IF NOT (Transfer.Mode = FIT_VFD_Transfer_Modes.Pause) AND NOT (Transfer.Mode = FIT_VFD_Transfer_Modes.Resume) THEN _w1 := Transfer.Mode; END_IF
Transfer.cONFIG.Mode_Memory := _w1;
IF Transfer.Mode = FIT_VFD_Transfer_Modes.Resume THEN _w2 := Transfer.Config.Mode_Memory; END_IF
Transfer.Mode := _w2;
Transfer.Status := SEL(VFD_Not_Ready, SEL(BCV_Not_Ready, SEL(ACV_Not_Ready, SEL(Transfer.Mode=FIT_VFD_Transfer_Modes.Lock_Out, SEL(False, SEL(Complete, SEL(Transfer_Running, SEL(FIT.PLC_Reset, SEL(IDLE_Return, SEL(PAUSED, Transfer_status.IDLE, Transfer_status.Paused), Transfer_status.IDLE), Transfer_status.FIT_Reset), Transfer_status.Running), Transfer_status.Complete), Transfer_status.Complete), Transfer_status.LOCKED_OUT), Transfer_status.ACV_Not_Ready), Transfer_status.BCV_Not_Ready), Transfer_status.VFD_Not_Ready);
_w3 := Transfer.Mode = FIT_VFD_Transfer_Modes.Idle;
_w4 := True AND NOT (BCV.Status = Burkert.eBCV_Status.A_Closed);
BCV_Not_Ready := _w3 AND _w4;
_w5 := True AND NOT (VFD.MODE.eMode = eVFD_Modes.Auto);
_w6 := _w4 OR _w5;
SR2(SET1 := _w3 AND _w6, RESET := NOT _w6); // SR
IF SR2.Q1 THEN _w7 := FIT_VFD_Transfer_Modes.Idle; END_IF
Transfer.Mode := _w7;
VFD_Not_Ready := _w3 AND _w5;
_w8 := Transfer.Status = Transfer_Status.Complete;
_w9 := Transfer.Status = Transfer_Status.BCV_Not_Ready OR Transfer.Status = Transfer_Status.VFD_Not_Ready;
_w10 := Transfer_Status.IDLE = Transfer.Status OR False OR Transfer.Status = Transfer_Status.LOCKED_OUT;
_w11 := Transfer.Mode = FIT_VFD_Transfer_Modes.Pause;
PAUSED := _w11;
_w12 := Transfer.Mode = FIT_VFD_Transfer_Modes.IDLE;
_w13 := Complete OR Error OR _w12 OR _w11;
_w14 := NOT Pump_Start OR _w13;
CTRL_PID_1(
    ACT := FIT.Rate,
    SET := Transfer.Config.Target_Rate,
    SUP := 0.0,
    OFS := Transfer.Config.Target_Rate * Transfer.Config.FF,
    M_I := 0.0,
    MAN := _w14,
    RST := _w14,
    KP := Transfer.Config.KP,
    TN := Transfer.Config.TN,
    TV := Transfer.Config.TV,
    LL := 0,
    LH := 100); // BURKERT_OSCAT_BASIC.CTRL_PID
PID_CV := CTRL_PID_1.Y;
TP11(IN := NOT LockOut_Active AND _w13, PT := t#5s); // TP
VFD.PLC_Run := SEL(TP11.Q, VFD.PLC_Run, FALSE);
VFD.PLC_CMD := SEL(TP11.Q, VFD.PLC_CMD, 0.0);
F_TRIG_0(CLK := TP11.Q); // F_Trig
BCV.PLC_CMD := SEL(F_TRIG_0.Q, BCV.PLC_CMD, False);
IDLE_Return := _w9 AND _w12;
SR_10(SET1 := FIT.Total<1, RESET := _w12); // SR
TON_10(IN := SR_10.Q1, PT := T#2s); // TON
FIT_Reset_Complete := TON_10.Q;
R_TRIG_0(CLK := _w12 OR TON_10.Q); // R_trig
_w15 := SEL(R_TRIG_0.Q, FIT.PLC_Reset, False);
_w16 := Transfer.Mode = FIT_VFD_Transfer_Modes.Batch;
_w17 := False OR False OR _w16;
Flow_Mode := _w17;
_w18 := _w17 AND FIT_Reset_Complete AND NOT Complete AND NOT Error AND NOT Time_Complete;
Transfer_Running := _w18;
transfer.Remaining_Volume := SEL(_w18, 0, Transfer.Config.Target_Volume-fit.Total);
_w19 := True AND _w18;
Enable_Pump := _w19;
BCV.PLC_CMD := SEL(_w19, BCV.PLC_CMD, TRUE);
_w20 := _w16 AND FIT_Reset_Complete AND FIT.Total >= Transfer.Config.Target_Volume;
Batch_Complete := _w20;
RS_11(SET := Time_Complete OR _w20 OR False, RESET1 := _w12); // RS
Complete := RS_11.Q1;
_w21 := LOCK_OUT AND _w10 AND NOT RS_11.Q1;
F_TRIG_10(CLK := _w21); // F_Trig
IF F_TRIG_10.Q THEN _w22 := FIT_VFD_Transfer_Modes.Idle; END_IF
Transfer.Mode := _w22;
_w23 := _w21;
IF _w23 THEN _w24 := FIT_VFD_Transfer_Modes.Lock_Out; END_IF
LockOut_Active := _w23;
Transfer.Mode := _w24;
FIT.PLC_Reset := SEL(NOT SR_10.Q1 AND _w17 AND NOT _w20, _w15, True);
_w25 := SEL(_w19, _w18, BCV.Status = Burkert.eBCV_Status.A_Open);
Pump_Start := _w25;
_w26 := SEL(_w25, VFD.PLC_CMD, PID_CV);
Transfer.Config.Motor_PCT := _w26;
VFD.PLC_CMD := _w26;
VFD.PLC_Run := SEL(_w25, VFD.PLC_Run, PID_CV > 15);
TON_12(IN := _w8, PT := T#10s); // TON

END_FUNCTION_BLOCK

// 25 Interfaces/IcSensorProvider
INTERFACE IcSensorProvider:

END_INTERFACE;

METHOD GetSensorRef : POINTER TO Burkert.cSensor
VAR_INPUT
        eSensor : cSensor_Mapping;
END_VAR
END_METHOD

END_INTERFACE

// 50 Functions/DaySeconds
FUNCTION DaySeconds : UDINT
VAR_INPUT
	Hour:UINT;
	Minute:UINT;
	Second:UINT;
END_VAR
VAR
END_VAR

(* body of a kind this reader does not render *)

END_FUNCTION

// GetLibVersion
// This function has been automatically generated from the project information.
FUNCTION GetLibVersion : VERSION
VAR_INPUT
	
END_VAR

GetLibVersion.uiMajor := 3;
GetLibVersion.uiMinor := 0;
GetLibVersion.uiServicePack := 0;
GetLibVersion.uiPatch := 49;

END_FUNCTION

// GetLibVersionNumber
// This function has been automatically generated from the project information.
FUNCTION GetLibVersionNumber : DWORD
VAR_INPUT
	
END_VAR

GetLibVersionNumber := 50331697;

END_FUNCTION

// IsLibReleased
// This function has been automatically generated from the project information.
FUNCTION IsLibReleased : BOOL
VAR_INPUT
	
END_VAR

IsLibReleased := FALSE;

END_FUNCTION

// GetBooleanProperty
// This function has been automatically generated from the project information.
{attribute 'signature_flag' := '1073741824'}
{attribute 'register_in_runtime'}
FUNCTION GetBooleanProperty : BOOL
VAR_INPUT
	stKey: WSTRING;
END_VAR

IF stKey = "IsEndUserLibrary" THEN
	GetBooleanProperty := FALSE;
ELSIF stKey = "IsStorageFormatPinned" THEN
	GetBooleanProperty := FALSE;
ELSIF stKey = "Released" THEN
	GetBooleanProperty := FALSE;
ELSE
	GetBooleanProperty := FALSE;
END_IF

END_FUNCTION

// GetCompany
// This function has been automatically generated from the project information.
{attribute 'signature_flag' := '1073741824'}
{attribute 'register_in_runtime'}
FUNCTION GetCompany : WSTRING
VAR_INPUT
	
END_VAR

GetCompany := "Burkert-Canada";

END_FUNCTION

// GetTextProperty2
// This function has been automatically generated from the project information.
{attribute 'signature_flag' := '1073741824'}
{attribute 'register_in_runtime'}
FUNCTION GetTextProperty2 : POINTER TO WSTRING
VAR_INPUT
	stKey: WSTRING;
END_VAR

IF stKey = "Author" THEN
	GetTextProperty2 := ADR("Robert Budgen");
ELSIF stKey = "Company" THEN
	GetTextProperty2 := ADR("Burkert-Canada");
ELSIF stKey = "CompiledLibraryCompatibilityVersion" THEN
	GetTextProperty2 := ADR("e!COCKPIT");
ELSIF stKey = "DefaultNamespace" THEN
	GetTextProperty2 := ADR("Brau");
ELSIF stKey = "Description" THEN
	GetTextProperty2 := ADR("");
ELSIF stKey = "LanguageModelAttribute" THEN
	GetTextProperty2 := ADR("qualified-access-only");
ELSIF stKey = "Placeholder" THEN
	GetTextProperty2 := ADR("Brau");
ELSIF stKey = "Project" THEN
	GetTextProperty2 := ADR("Burkert Canada");
ELSIF stKey = "Title" THEN
	GetTextProperty2 := ADR("Brau");
ELSE
	GetTextProperty2 := ADR("");
END_IF

END_FUNCTION

// GetTextProperty
// This function has been automatically generated from the project information.
{attribute 'signature_flag' := '1073741824'}
{attribute 'register_in_runtime'}
FUNCTION GetTextProperty : WSTRING
VAR_INPUT
	stKey: WSTRING;
END_VAR

IF stKey = "Author" THEN
	GetTextProperty := "Robert Budgen";
ELSIF stKey = "Company" THEN
	GetTextProperty := "Burkert-Canada";
ELSIF stKey = "CompiledLibraryCompatibilityVersion" THEN
	GetTextProperty := "e!COCKPIT";
ELSIF stKey = "DefaultNamespace" THEN
	GetTextProperty := "Brau";
ELSIF stKey = "Description" THEN
	GetTextProperty := "";
ELSIF stKey = "LanguageModelAttribute" THEN
	GetTextProperty := "qualified-access-only";
ELSIF stKey = "Placeholder" THEN
	GetTextProperty := "Brau";
ELSIF stKey = "Project" THEN
	GetTextProperty := "Burkert Canada";
ELSIF stKey = "Title" THEN
	GetTextProperty := "Brau";
ELSE
	GetTextProperty := "";
END_IF

END_FUNCTION

// GetTitle
// This function has been automatically generated from the project information.
{attribute 'signature_flag' := '1073741824'}
{attribute 'register_in_runtime'}
FUNCTION GetTitle : WSTRING
VAR_INPUT
	
END_VAR

GetTitle := "Brau";

END_FUNCTION

// GetVersion
// This function has been automatically generated from the project information.
{attribute 'signature_flag' := '1073741824'}
{attribute 'register_in_runtime'}
FUNCTION GetVersion : VERSION
VAR_INPUT
	
END_VAR

GetVersion.uiMajor := 3;
GetVersion.uiMinor := 0;
GetVersion.uiServicePack := 0;
GetVersion.uiPatch := 49;

END_FUNCTION

// GetVersionProperty
// This function has been automatically generated from the project information.
{attribute 'signature_flag' := '1073741824'}
{attribute 'register_in_runtime'}
FUNCTION GetVersionProperty : VERSION
VAR_INPUT
	stKey: WSTRING;
END_VAR

IF stKey = "Version" THEN
	GetVersionProperty.uiMajor := 3;
	GetVersionProperty.uiMinor := 0;
	GetVersionProperty.uiServicePack := 0;
	GetVersionProperty.uiPatch := 49;
ELSE
	GetVersionProperty.uiMajor := 0;
	GetVersionProperty.uiMinor := 0;
	GetVersionProperty.uiServicePack := 0;
	GetVersionProperty.uiPatch := 0;
END_IF

END_FUNCTION

// Asi/AC2916_AIT
FUNCTION_BLOCK AC2916_AIT
VAR_INPUT
	//Raw:	REAL;
	LAS:BOOL:=TRUE;
	LDS:BOOL:=TRUE;
	LPS:BOOL:=TRUE;
	LPF:BOOL:=FALSE;
	Alarm_Enable:BOOL:=TRUE;
	Latching:BOOL:=FALSE;
	//Fault:BOOL:=FALSE;
	Online:BOOL:=TRUE;
	Raw:WORD;
END_VAR

VAR_OUTPUT
	//Status	:BYTE;
END_VAR
VAR_IN_OUT
AIT	:	Burkert.cAIT;
END_VAR

VAR
	hihi: BOOL;
	hi: BOOL;
	lolo: BOOL;
	LO: BOOL;
	Alarm_Debounce: TON;
	deboune_Time: TIME;
	Alarm_Active: BOOL;
	Alarm_Debounce_ET: TIME;
	Alarm: BOOL;
	ALARM_2_0: BURKERT_OSCAT_BASIC.ALARM_2;
	F_TRIG_0: F_Trig;
	TON_0: TON;
	tmpEU: REAL;
	//tmpEU1: REAL;
	tmpEU2: REAL;
END_VAR

VAR_TEMP
	EU_Range: REAL;
	Raw_Range: REAL;
	Corrected_Raw: REAL;
	Raw_Pct: REAL;
	EU_Scaled: REAL;
END_VAR
VAR // added by the converter: edge detectors and wires of the graphical bodies
    _w1, _w2, _w3 : BOOL;
END_VAR

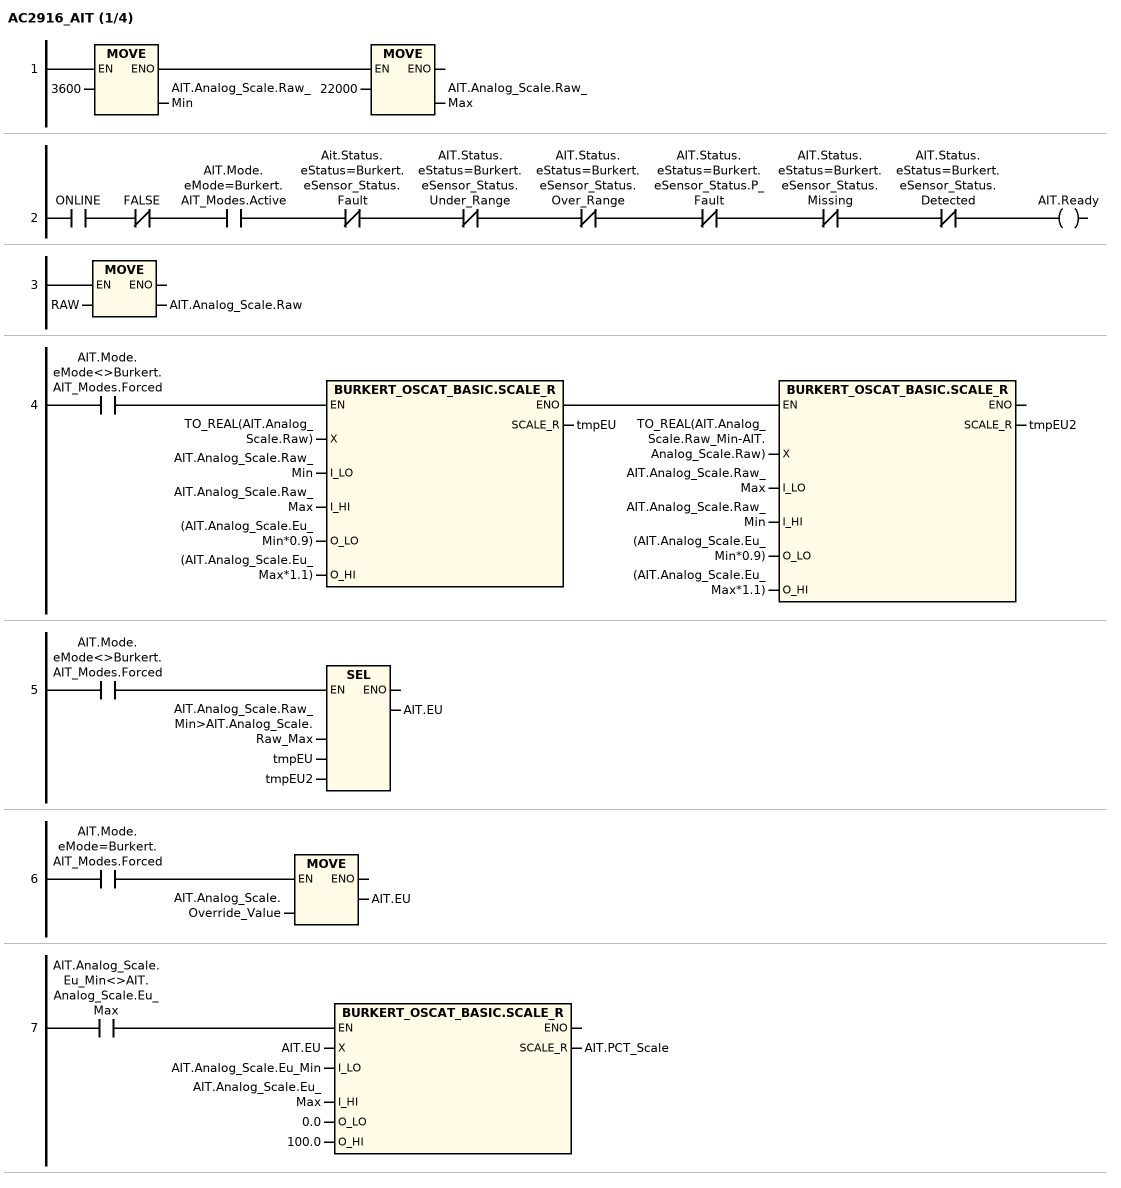
// NETWORK 1
AIT.Analog_Scale.Raw_Min := 3600;
AIT.Analog_Scale.Raw_Max := 22000;

// NETWORK 2
AIT.Ready := ONLINE AND NOT FALSE AND (AIT.Mode.eMode=Burkert.AIT_Modes.Active) AND NOT (Ait.Status.eStatus=Burkert.eSensor_Status.Fault) AND NOT (AIT.Status.eStatus=Burkert.eSensor_Status.Under_Range) AND NOT (AIT.Status.eStatus=Burkert.eSensor_Status.Over_Range) AND NOT (AIT.Status.eStatus=Burkert.eSensor_Status.P_Fault) AND NOT (AIT.Status.eStatus=Burkert.eSensor_Status.Missing) AND NOT (AIT.Status.eStatus=Burkert.eSensor_Status.Detected);

// NETWORK 3
AIT.Analog_Scale.Raw := RAW;

// NETWORK 4
_w1 := AIT.Mode.eMode<>Burkert.AIT_Modes.Forced;
IF _w1 THEN
    tmpEU := BURKERT_OSCAT_BASIC.SCALE_R(X := TO_REAL(AIT.Analog_Scale.Raw), I_LO := AIT.Analog_Scale.Raw_Min, I_HI := AIT.Analog_Scale.Raw_Max, O_LO := (AIT.Analog_Scale.Eu_Min*0.9), O_HI := (AIT.Analog_Scale.Eu_Max*1.1));
END_IF
IF _w1 THEN
    tmpEU2 := BURKERT_OSCAT_BASIC.SCALE_R(X := TO_REAL(AIT.Analog_Scale.Raw_Min-AIT.Analog_Scale.Raw), I_LO := AIT.Analog_Scale.Raw_Max, I_HI := AIT.Analog_Scale.Raw_Min, O_LO := (AIT.Analog_Scale.Eu_Min*0.9), O_HI := (AIT.Analog_Scale.Eu_Max*1.1));
END_IF

// NETWORK 5
IF AIT.Mode.eMode<>Burkert.AIT_Modes.Forced THEN
    AIT.EU := SEL(AIT.Analog_Scale.Raw_Min>AIT.Analog_Scale.Raw_Max, tmpEU, tmpEU2);
END_IF

// NETWORK 6
IF AIT.Mode.eMode=Burkert.AIT_Modes.Forced THEN AIT.EU := AIT.Analog_Scale.Override_Value; END_IF

// NETWORK 7
IF AIT.Analog_Scale.Eu_Min<>AIT.Analog_Scale.Eu_Max THEN
    AIT.PCT_Scale := BURKERT_OSCAT_BASIC.SCALE_R(X := AIT.EU, I_LO := AIT.Analog_Scale.Eu_Min, I_HI := AIT.Analog_Scale.Eu_Max, O_LO := 0.0, O_HI := 100.0);
END_IF

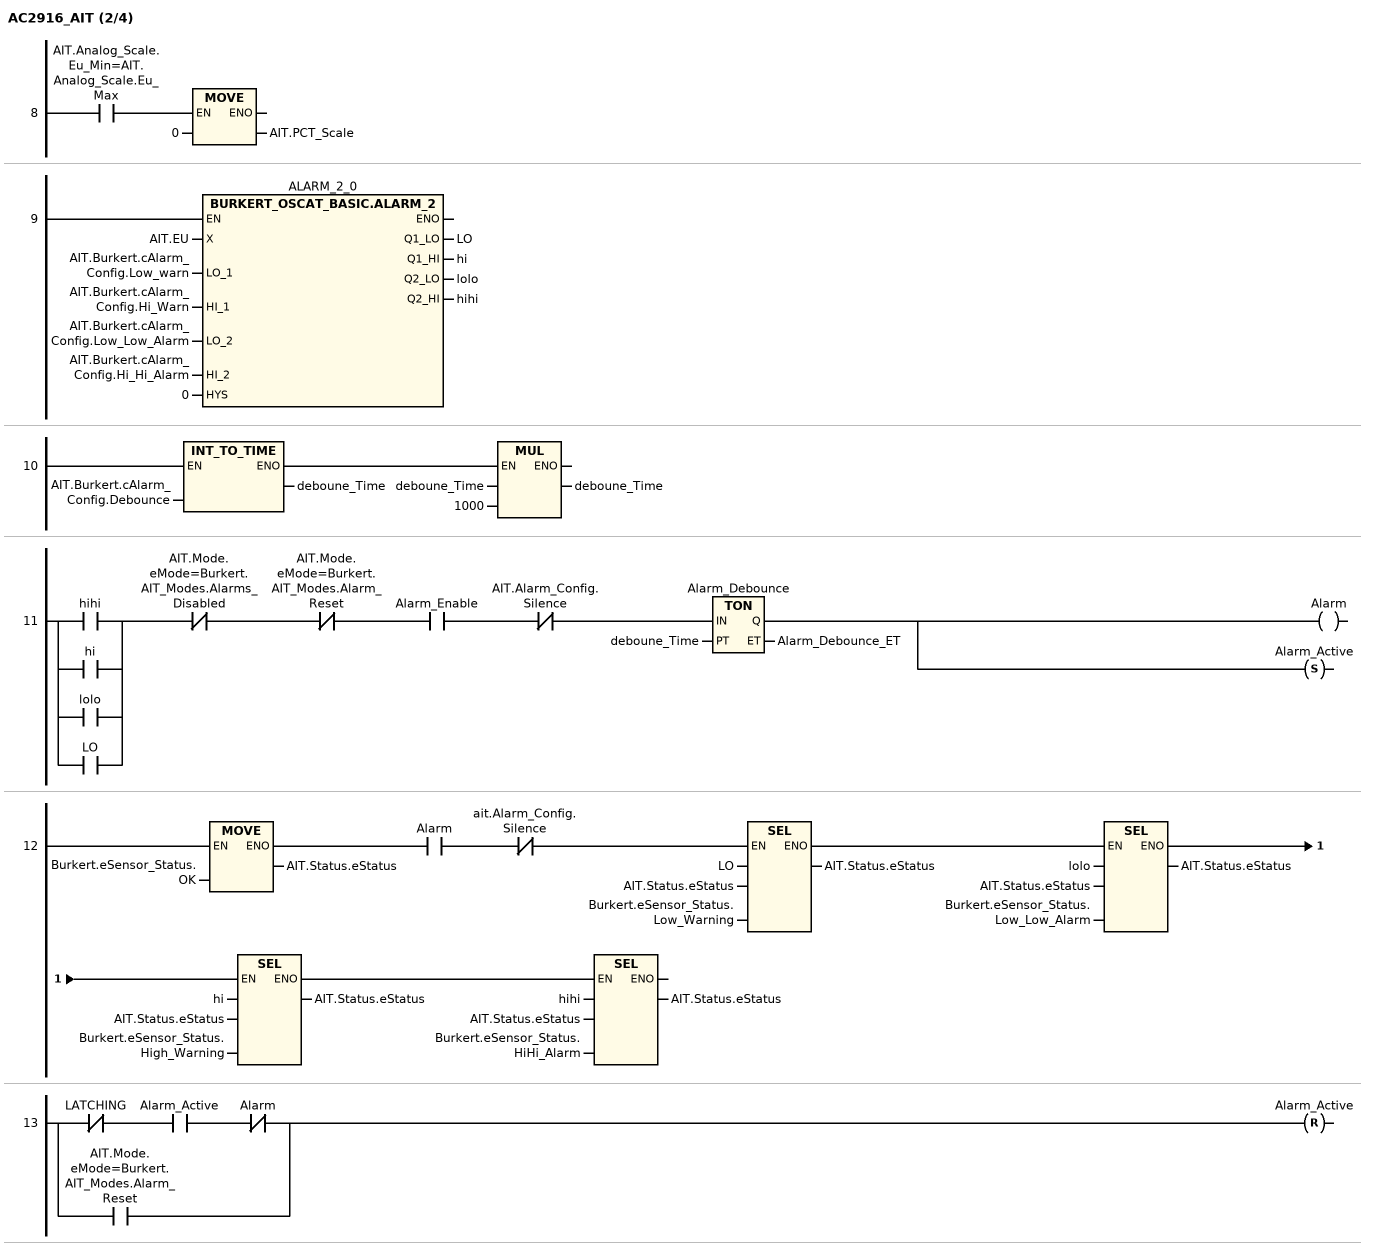
// NETWORK 8
IF AIT.Analog_Scale.Eu_Min=AIT.Analog_Scale.Eu_Max THEN AIT.PCT_Scale := 0; END_IF

// NETWORK 9
ALARM_2_0(
    X := AIT.EU,
    LO_1 := AIT.Burkert.cAlarm_Config.Low_warn,
    HI_1 := AIT.Burkert.cAlarm_Config.Hi_Warn,
    LO_2 := AIT.Burkert.cAlarm_Config.Low_Low_Alarm,
    HI_2 := AIT.Burkert.cAlarm_Config.Hi_Hi_Alarm,
    HYS := 0,
    Q1_LO => LO,
    Q1_HI => hi,
    Q2_LO => lolo,
    Q2_HI => hihi); // BURKERT_OSCAT_BASIC.ALARM_2

// NETWORK 10
deboune_Time := INT_TO_TIME(AIT.Burkert.cAlarm_Config.Debounce);
deboune_Time := deboune_Time * 1000;

// NETWORK 11
Alarm_Debounce(
    IN := (hihi OR hi OR lolo OR LO) AND NOT (AIT.Mode.eMode=Burkert.AIT_Modes.Alarms_Disabled) AND NOT (AIT.Mode.eMode=Burkert.AIT_Modes.Alarm_Reset) AND Alarm_Enable AND NOT AIT.Alarm_Config.Silence,
    PT := deboune_Time,
    ET => Alarm_Debounce_ET); // TON
Alarm := Alarm_Debounce.Q;
Alarm_Active S= Alarm_Debounce.Q;

// NETWORK 12
AIT.Status.eStatus := Burkert.eSensor_Status.OK;
_w2 := Alarm AND NOT ait.Alarm_Config.Silence;
IF _w2 THEN AIT.Status.eStatus := SEL(LO, AIT.Status.eStatus, Burkert.eSensor_Status.Low_Warning); END_IF
IF _w2 THEN AIT.Status.eStatus := SEL(lolo, AIT.Status.eStatus, Burkert.eSensor_Status.Low_Low_Alarm); END_IF
IF _w2 THEN AIT.Status.eStatus := SEL(hi, AIT.Status.eStatus, Burkert.eSensor_Status.High_Warning); END_IF
IF _w2 THEN AIT.Status.eStatus := SEL(hihi, AIT.Status.eStatus, Burkert.eSensor_Status.HiHi_Alarm); END_IF

// NETWORK 13
Alarm_Active R= NOT LATCHING AND Alarm_Active AND NOT Alarm OR (AIT.Mode.eMode=Burkert.AIT_Modes.Alarm_Reset);

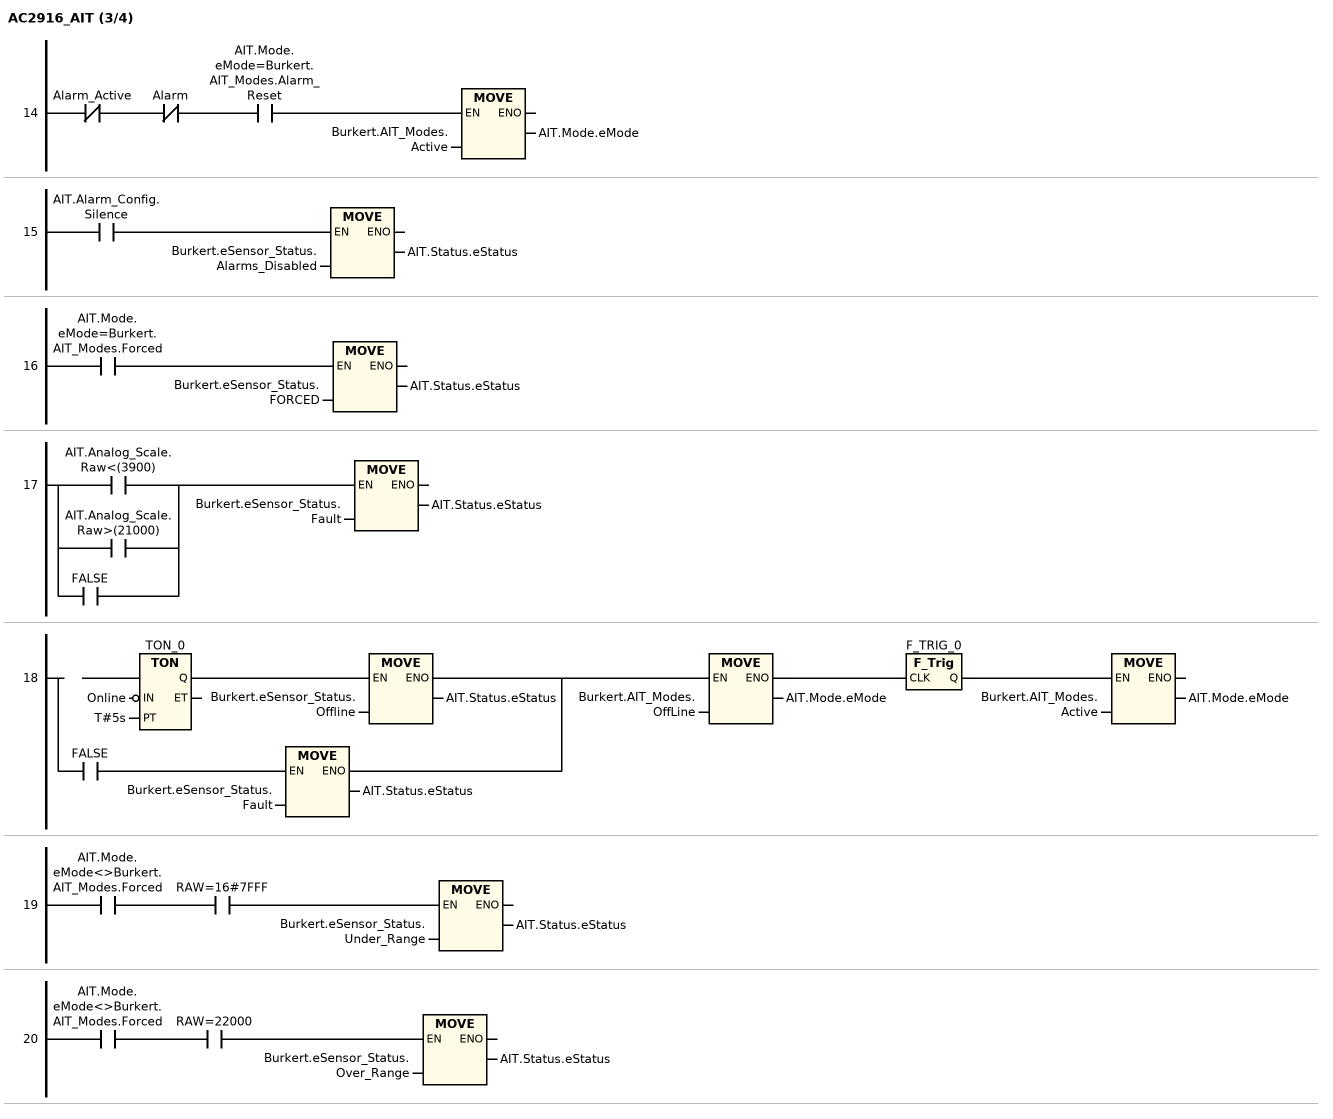
// NETWORK 14
IF NOT Alarm_Active AND NOT Alarm AND (AIT.Mode.eMode=Burkert.AIT_Modes.Alarm_Reset) THEN
    AIT.Mode.eMode := Burkert.AIT_Modes.Active;
END_IF

// NETWORK 15
IF AIT.Alarm_Config.Silence THEN AIT.Status.eStatus := Burkert.eSensor_Status.Alarms_Disabled; END_IF

// NETWORK 16
IF AIT.Mode.eMode=Burkert.AIT_Modes.Forced THEN AIT.Status.eStatus := Burkert.eSensor_Status.FORCED; END_IF

// NETWORK 17
IF (AIT.Analog_Scale.Raw<(3900)) OR (AIT.Analog_Scale.Raw>(21000)) OR FALSE THEN
    AIT.Status.eStatus := Burkert.eSensor_Status.Fault;
END_IF

// NETWORK 18
TON_0(IN := NOT Online, PT := T#5s); // TON
_w3 := TON_0.Q;
IF _w3 THEN AIT.Status.eStatus := Burkert.eSensor_Status.Offline; END_IF
IF FALSE THEN AIT.Status.eStatus := Burkert.eSensor_Status.Fault; END_IF
IF _w3 OR FALSE THEN AIT.Mode.eMode := Burkert.AIT_Modes.OffLine; END_IF
F_TRIG_0(CLK := _w3 OR FALSE); // F_Trig
IF F_TRIG_0.Q THEN AIT.Mode.eMode := Burkert.AIT_Modes.Active; END_IF

// NETWORK 19
IF (AIT.Mode.eMode<>Burkert.AIT_Modes.Forced) AND (RAW=16#7FFF) THEN
    AIT.Status.eStatus := Burkert.eSensor_Status.Under_Range;
END_IF

// NETWORK 20
IF (AIT.Mode.eMode<>Burkert.AIT_Modes.Forced) AND (RAW=22000) THEN
    AIT.Status.eStatus := Burkert.eSensor_Status.Over_Range;
END_IF

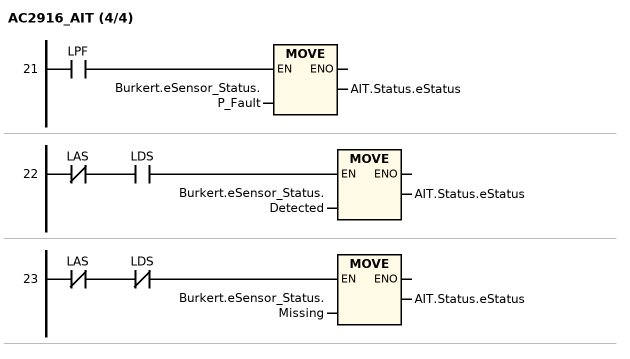
// NETWORK 21
IF LPF THEN AIT.Status.eStatus := Burkert.eSensor_Status.P_Fault; END_IF

// NETWORK 22
IF NOT LAS AND LDS THEN AIT.Status.eStatus := Burkert.eSensor_Status.Detected; END_IF

// NETWORK 23
IF NOT LAS AND NOT LDS THEN AIT.Status.eStatus := Burkert.eSensor_Status.Missing; END_IF

END_FUNCTION_BLOCK

// Asi/ACV_ASI_CTRL_UDFB
FUNCTION_BLOCK ACV_ASI_CTRL_UDFB
VAR_INPUT
	FB:INT;
	CutOff:REAL:=0;
	LOCKOUT:BOOL:=FALSE;
	Online:BOOL:=TRUE;
	Error_PCT:REAL:=10;
	Error_Delay_S:INT:=10;
	LAS:BOOL:=TRUE;
	LDS:BOOL:=TRUE;
	LPS:BOOL:=TRUE;
	LPF:BOOL:=FALSE;
END_VAR
VAR_OUTPUT
	Status	:INT;
	Output	:INT;
END_VAR
VAR_IN_OUT
	//Valve	:ACV_DUT;
END_VAR
VAR
	//Output_TMP: REAL;
	//Scaled_Out: REAL;
	TON_1: TON;
	TOF_0: TOF;
	tmp_Output: REAL;
	FB_Real: REAL;
	Burkert_mode: Ton;
END_VAR

VAR_IN_OUT
	Valve:Burkert.ASi_8694;
END_VAR

(* body of a kind this reader does not render *)

END_FUNCTION_BLOCK

// Asi/B8681_ASI_UDFB
FUNCTION_BLOCK B8681_ASI_UDFB
VAR_INPUT
	RX:BYTE;
	LAS:BOOL:=TRUE;
	LDS:BOOL:=TRUE;
	LPS:BOOL:=TRUE;
	LPF:BOOL:=FALSE;
END_VAR
VAR_OUTPUT
	TX:BYTE;
END_VAR
VAR
	lcl_status: BYTE;
END_VAR
VAR_IN_OUT
	Valve:Burkert.B8691_Asi_DUT;
END_VAR
VAR // added by the converter: edge detectors and wires of the graphical bodies
    _w1, _w2, _w3 : ANY;
END_VAR

_w1 := (Valve.Mode=Burkert.e_8681_Modes.Auto) AND (Valve.PLC_CMD=Burkert.e_8681_Modes.Upper_Drain) OR (Valve.Mode=Burkert.e_8681_Modes.Upper_Drain);
_w2 := SEL(_w1, SEL((Valve.Mode=Burkert.e_8681_Modes.Auto) AND (Valve.PLC_CMD=Burkert.e_8681_Modes.Lower_Drain) OR (Valve.Mode=Burkert.e_8681_Modes.Lower_Drain), SEL((Valve.Mode=Burkert.e_8681_Modes.Auto) AND (Valve.PLC_CMD=Burkert.e_8681_Modes.Open) OR (Valve.Mode=Burkert.e_8681_Modes.Open), 0, 1), 2), 4);
TX := _w2;
BURKERT_OSCAT_BASIC.WORD_OF_BYTE\(B1 := _w2, B0 := RX, WORD_OF_BYTE => _w3);
Valve.Status := _w3;
Valve.Status1 := SEL(LPF, SEL(LDS AND NOT LAS, SEL(NOT LAS, SEL(RX.2, SEL(_w1, SEL(RX.0, SEL(RX.1, eB8681_Status.Unknown, eB8681_Status.Open), eB8681_Status.Blocked), eB8681_Status.Upper_Drain), eB8681_Status.Lower_Drain), eB8681_Status.Missing), eB8681_Status.Detected), eB8681_Status.P_Fault);

END_FUNCTION_BLOCK

// Asi/BCV_ASI_CTRL_UDFB
FUNCTION_BLOCK BCV_ASI_CTRL_UDFB
VAR_INPUT
	OL:BOOL;
	CL:BOOL;
	LOCKOUT:BOOL:=FALSE;
	Online:BOOL:=TRUE;
	LAS:BOOL:=TRUE;
	LDS:BOOL:=TRUE;
	LPS:BOOL:=TRUE;
	LPF:BOOL:=FALSE;

END_VAR
VAR_OUTPUT
	Output	:BOOL;
END_VAR
VAR_IN_OUT
	BCV:Burkert.cBCV;
END_VAR
VAR
	
	Test: BOOL;
	GEN_PULSE_0: Burkert_OSCAT_BASIC.GEN_PULSE;
	Burkert_Open_Ton: TON;
END_VAR

(* body of a kind this reader does not render *)

END_FUNCTION_BLOCK

// Burkert Library/Parse_DDO
FUNCTION_BLOCK Parse_DDO
VAR_INPUT
	ORF_data:POINTER TO BYTE;
	Node:BYTE;
	Request_Size:INT:=10;
	
END_VAR
VAR_OUTPUT
	DDO:eDip_DDO;
END_VAR
VAR
	Block_Size:UINT;
	lcl_pointer:POINTER TO BYTE;
	DDO_Index:INT;
	ORF_Node:BYTE;
	ORF_Index_HB:BYTE;
	ORF_Index_LB:BYTE;
	ORF_SubIndex:BYTE;
	
	
END_VAR

Block_Size:=SIZEOF(ORF_Request);
lcl_pointer:=ORF_Data;

FOR DDO_Index := 0 TO Request_Size BY 1 DO
	
	ORF_Index_LB:=lcl_pointer[0];
	ORF_Index_HB:=LCL_Pointer[1];
	ORF_SubIndex:=lcl_pointer[2];
	ORF_Node:=lcl_pointer[3];
	
	
	IF (lcl_pointer[10]=1) AND (ORF_Node= Node) AND (ORF_Index_HB=16#20) AND (ORF_Index_LB=16#00) THEN
		MEMUtils.MemSet(pbyBuffer:=lcl_pointer+10 , byValue:=0 , dwSize:= 1); // Clear Complete
		CASE ORF_SubIndex OF
			16#02: //16#2000-2
				MEMUtils.MemCpy(pbyDest:=ADR(DDO.Ident)+2 , pbySrc:=lcl_pointer+4 , dwSize:=2 );
				MEMUtils.MemCpy(pbyDest:=ADR(DDO.Ident) , pbySrc:=lcl_pointer+6 , dwSize:=2 );
				lcl_pointer[9]:=BOOL_TO_BYTE(DDO.Ident=0);
				//MEMUtils.MemSet(pbyBuffer:=lcl_pointer+9 , byValue:=1 , dwSize:= 1);// Set Enable				
			16#07: //16#2000-7
				MEMUtils.MemCpy(pbyDest:=ADR(DDO.Serial)+2 , pbySrc:=lcl_pointer+4 , dwSize:=2 );
				MEMUtils.MemCpy(pbyDest:=ADR(DDO.Serial) , pbySrc:=lcl_pointer+6 , dwSize:=2 );
				lcl_pointer[9]:=BOOL_TO_BYTE(DDO.Serial=0);
			16#008: //16#2000-8
				MEMUtils.MemCpy(pbyDest:=ADR(DDO.Product_Code)+2 , pbySrc:=lcl_pointer+4 , dwSize:=2 );
				MEMUtils.MemCpy(pbyDest:=ADR(DDO.Product_Code) , pbySrc:=lcl_pointer+6 , dwSize:=2 );
				lcl_pointer[9]:=BOOL_TO_BYTE(DDO.Product_Code =0);
		END_CASE;	
	END_IF;
	lcl_pointer:=lcl_pointer+Block_Size;
END_FOR;

END_FUNCTION_BLOCK

// Burkert Library/Parse_DSO
FUNCTION_BLOCK Parse_DSO
VAR_INPUT
	ORF_data:POINTER TO BYTE;
	Node:BYTE;
	Request_Size:INT:=10;
	
END_VAR
VAR_OUTPUT
	DSO:eDip_DSO;
END_VAR
VAR
	Block_Size:UINT;
	lcl_pointer:POINTER TO BYTE;
	DSO_Index:INT;
	ORF_Node:BYTE;
	ORF_Index_HB:BYTE;
	ORF_Index_LB:BYTE;
	ORF_SubIndex:BYTE;
	
END_VAR

Block_Size:=SIZEOF(ORF_Request);
lcl_pointer:=ORF_Data;

FOR DSO_Index := 0 TO Request_Size BY 1 DO
	ORF_Index_LB:=lcl_pointer[0];
	ORF_Index_HB:=LCL_Pointer[1];
	ORF_SubIndex:=lcl_pointer[2];
	ORF_Node:=lcl_pointer[3];
	
	IF (lcl_pointer[10]=1) AND (ORF_Node= Node) AND (ORF_Index_HB=16#20) AND (ORF_Index_LB=16#04) THEN
		//MEMUtils.MemSet(pbyBuffer:=lcl_pointer+10 , byValue:=0 , dwSize:= 1); // Clear Complete
		lcl_pointer[10]:=0;
		CASE ORF_SubIndex OF
			
			16#01: //16#2004-1
				MEMUtils.MemCpy(pbyDest:=ADR(DSO.NamurNe107) , pbySrc:=lcl_pointer+6 , dwSize:=1 );
				//MEMUtils.MemSet(pbyBuffer:=lcl_pointer+9 , byValue:=1 , dwSize:= 1);// Set Enable
				lcl_pointer[9]:=1;
			16#02: //16#2004-2
				MEMUtils.MemCpy(pbyDest:=ADR(DSO.Temperature)+2 , pbySrc:=lcl_pointer+4 , dwSize:=2 );
				MEMUtils.MemCpy(pbyDest:=ADR(DSO.Temperature) , pbySrc:=lcl_pointer+6 , dwSize:=2 );
				//MEMUtils.MemSet(pbyBuffer:=lcl_pointer+9 , byValue:=1 , dwSize:= 1);// Set Enable
				lcl_pointer[9]:=1;
			16#03: //16#2004-3
				MEMUtils.MemCpy(pbyDest:=ADR(DSO.Voltage)+2 , pbySrc:=lcl_pointer+4 , dwSize:=2 );
				MEMUtils.MemCpy(pbyDest:=ADR(DSO.Voltage) , pbySrc:=lcl_pointer+6 , dwSize:=2 );
				//MEMUtils.MemSet(pbyBuffer:=lcl_pointer+9 , byValue:=1 , dwSize:= 1);// Set Enable
				lcl_pointer[9]:=1;
			16#04: //16#2004-4
				MEMUtils.MemCpy(pbyDest:=ADR(DSO.Operational_Time_S)+2 , pbySrc:=lcl_pointer+4 , dwSize:=2 );
				MEMUtils.MemCpy(pbyDest:=ADR(DSO.Operational_Time_S) , pbySrc:=lcl_pointer+6 , dwSize:=2 );
				//MEMUtils.MemSet(pbyBuffer:=lcl_pointer+9 , byValue:=1 , dwSize:= 1);// Set Enable
				lcl_pointer[9]:=1;
			16#05: //16#2004-5
				MEMUtils.MemCpy(pbyDest:=ADR(DSO.Max_Temp)+2 , pbySrc:=lcl_pointer+4 , dwSize:=2 );
				MEMUtils.MemCpy(pbyDest:=ADR(DSO.Max_Temp) , pbySrc:=lcl_pointer+6 , dwSize:=2 );
				//MEMUtils.MemSet(pbyBuffer:=lcl_pointer+9 , byValue:=1 , dwSize:= 1);// Set Enable
				lcl_pointer[9]:=1;
			16#06: //16#2004-6
				MEMUtils.MemCpy(pbyDest:=ADR(DSO.Min_Temp)+2 , pbySrc:=lcl_pointer+4 , dwSize:=2 );
				MEMUtils.MemCpy(pbyDest:=ADR(DSO.Min_Temp) , pbySrc:=lcl_pointer+6 , dwSize:=2 );
				//MEMUtils.MemSet(pbyBuffer:=lcl_pointer+9 , byValue:=1 , dwSize:= 1);// Set Enable
				lcl_pointer[9]:=1;
			16#07: //16#2004-7
				MEMUtils.MemCpy(pbyDest:=ADR(DSO.Max_Voltage)+2 , pbySrc:=lcl_pointer+4 , dwSize:=2 );
				MEMUtils.MemCpy(pbyDest:=ADR(DSO.Max_Voltage) , pbySrc:=lcl_pointer+6 , dwSize:=2 );
				//MEMUtils.MemSet(pbyBuffer:=lcl_pointer+9 , byValue:=1 , dwSize:= 1);// Set Enable
				lcl_pointer[9]:=1;
			16#08: //16#2004-8
				MEMUtils.MemCpy(pbyDest:=ADR(DSO.Min_Voltage)+2 , pbySrc:=lcl_pointer+4 , dwSize:=2 );
				MEMUtils.MemCpy(pbyDest:=ADR(DSO.Min_Voltage) , pbySrc:=lcl_pointer+6 , dwSize:=2 );
				//MEMUtils.MemSet(pbyBuffer:=lcl_pointer+9 , byValue:=1 , dwSize:= 1);// Set Enable
				lcl_pointer[9]:=1;
		END_CASE;	
	END_IF;
	lcl_pointer:=lcl_pointer+Block_Size;
END_FOR;

END_FUNCTION_BLOCK

// FB_PositionTracker
FUNCTION_BLOCK FB_PositionTracker
VAR_IN_OUT
    Position : REAL;   // Live position to be tracked
END_VAR

VAR_INPUT
    Count : REAL;      // Encoder count input
    FWD   : BOOL;      // Motor forward signal
    REV   : BOOL;      // Motor reverse signal
	
END_VAR

VAR
    LastCount : REAL;  // Previous encoder count
    Delta     : REAL;  // Change in count
END_VAR

IF Count<>Count THEN Count:=0; END_IF;



IF (FWD OR REV) THEN
    Delta := Count - LastCount;
    IF FWD THEN
        Position := Position + Delta;
    ELSIF REV THEN
        Position := Position - Delta;
    END_IF;
END_IF;

LastCount := Count;

END_FUNCTION_BLOCK

// fbMidPoint
FUNCTION fbMidPoint : REAL
VAR_INPUT
	LOW:REAL;
	High:REAL;
END_VAR
VAR
END_VAR

fbMidPoint:=(
	LOW+((High-LOW)/2)
);

END_FUNCTION

// RCP_Manager
FUNCTION RCP_Manager

VAR_IN_OUT
	Save:BOOL;
	Load:BOOL;
		Loaded:BOOL;
	Count:UINT;
END_VAR
VAR_OUTPUT

END_VAR
VAR
	RecipeManCommands:RecipeManCommands;
	Save_Response:DWORD;
	Load_Response:DWORD;
	Storage_Response:Bool;
	Load_Ton:ton;
	Save_Ton:Ton;
	Auto_Load_Ton:Ton;
	File_Save:BOOL;
	File_Save_Response:DWORD;
	//RCP_Names:ARRAY[0..9] OF STRING;
	
END_VAR
VAR
	R_Trig_0: R_Trig;
	Save_R_trig:R_trig;
END_VAR

RecipeManCommands();
Storage_Response:=RecipeManCommands.SetStoragePath('RCP/');
//RecipeManCommands.GetRecipeNames(RecipeDefinitionName:='PersistentVariables',pStrings:=ADR(RCP_Names),iSize:=10,iStartIndex:=0);
Save_R_trig(CLK:=Save);
IF Save_R_trig.Q THEN Save_Response:=16#FFFF; END_IF;


IF Save THEN 
	//Save_Response:=16#FFFF;	
	Save_Response:=ReadAndSave();
	END_IF;
IF Load THEN	Load_Response:=LoadAndWrite(); END_IF;


Save_ton(In:=Save AND NOT(Save_Response=16#FFFF),PT:=T#2S);
IF Save_Ton.Q THEN Save:=FALSE; END_IF;




Load_ton(In:=Load,PT:=T#2S);
IF Load_Ton.Q THEN		
	Load :=FALSE;
	Loaded:=TRUE;
	END_IF;

Auto_Load_Ton(IN:=NOT(Loaded),PT:=T#5S);

IF Auto_load_Ton.Q THEN Load:=TRUE;	END_IF;
//IF GVL.Day_Seconds=30500 THEN GVL.RCP_Save:=TRUE; END_IF;

R_Trig_0(CLK:=Save);
IF R_Trig_0.Q THEN	Count:=Count+1;	END_IF;



//IF File_Save THEN 
	//File_Save_Response:=RecipeManCommands.SaveRecipe	(RecipeDefinitionName:='PersistentVariables',RecipeName:='Day_27');//,FileName:='BackUp_1.txtrecipe'); 
//END_IF;

END_FUNCTION

// Virtual_FIT
FUNCTION_BLOCK Virtual_FIT
VAR
	Old_Total: REAL;
	OLD_V_Total: REAL;
	F_TRIG_0: F_trig;
	R_TRIG_0: R_trig;
END_VAR

VAR_OUTPUT
	V_Total:REAL;
END_VAR

VAR_INPUT
	Active:BOOL;
	Reset:BOOL;
	Total_IN:REAL;
END_VAR
VAR // added by the converter: edge detectors and wires of the graphical bodies
    _w1 : BOOL;
    _w2, _w3, _w4, _w5 : REAL;
    _w6 : ANY;
END_VAR

_w1 := Active AND (Total_In>0);
R_TRIG_0(CLK := (Total_In=0) AND Active); // R_trig
_w2 := SEL(_w1, Total_In, SEL(R_TRIG_0.Q, Old_Total, 0.0));
_w3 := SEL(_w2 >= 0.0, 0.0, _w2);
Old_Total := _w3;
_w4 := Total_In - _w3;
F_TRIG_0(CLK := Active); // F_trig
IF F_TRIG_0.Q OR Reset THEN _w5 := V_Total; END_IF
OLD_V_Total := _w5;
V_Total := _w4 + SEL(Reset, _w5, 0.0);
IF Reset THEN _w6 := 0.0; END_IF
OLD_V_Total := _w6;

END_FUNCTION_BLOCK

// Level_0_Remote_IO/AL1340_UDFB
FUNCTION_BLOCK AL1340_UDFB
VAR
	i:INT;
	msgCounter:BYTE;
END_VAR


VAR_INPUT
	//Acyclic_Response:cIFM_AL1342_Acyclic_Response;
	Device:	REFERENCE TO cIFM_AL1340;
END_VAR


VAR_OUTPUT
	//Port_Response:ARRAY[1..4] OF cIFM_AL1342_Acyclic_Response;
	//Acyclic_Request:cIFM_AL1342_Acyclic_Request;
	//Acyclic_Request_Active:BOOL;
END_VAR
VAR_IN_OUT
	//Port_Request:ARRAY[1..4] OF cIFM_AL1342_Acyclic_Request;
END_VAR


(*

IF Acyclic_Response.Port>0 THEN
	Port_Response[Acyclic_Response.Port]:=Acyclic_Response;
	Port_Response[Acyclic_Response.Port].Port:=0;
	
END_IF;

IF Port_Request[i+1].Port =16#FF THEN
	msgCounter:=msgCounter+1;
	Port_Request[i+1].Port:=TO_WORD(i+1);
	Port_Request[i+1].User_ID:=msgCounter;
	Acyclic_Request:=Port_Request[i+1];
	Acyclic_Request_Active:=TRUE;
	
ELSE
	i:=(i+1) MOD 8;	
	Acyclic_Request_Active:=FALSE;
END_IF;

*)

IF 	Device.Response.Port>0 THEN
	Device.Port_Response[Device.Response.Port]:=device.Response;
	Device.Port_Response[Device.Response.Port].Port:=0;
	
END_IF;

//Device.Port_Request
IF Device.Port_Request[i+1].Port =16#FF THEN
	msgCounter:=msgCounter+1;
	Device.Port_Request[i+1].Port:=TO_WORD(i+1);
	Device.Port_Request[i+1].User_ID:=msgCounter;
	Device.Request:=Device.Port_Request[i+1];
	Device.Acyclic_Request:=TRUE;
	
ELSE
	i:=(i+1) MOD 4;	
	Device.Acyclic_Request:=FALSE;
END_IF;

END_FUNCTION_BLOCK

// Level_0_Remote_IO/AL1342_UDFB
FUNCTION_BLOCK AL1342_UDFB
VAR
	i:INT;
	msgCounter:BYTE;
END_VAR

VAR_INPUT
	Response:cIFM_AL1342_Acyclic_Response;
	
END_VAR


VAR_OUTPUT
	Port_Response:ARRAY[1..8] OF cIFM_AL1342_Acyclic_Response;
	Request:cIFM_AL1342_Acyclic_Request;
	Acyclic_Request:BOOL;
END_VAR
VAR_IN_OUT
	Port_Request:ARRAY[1..8] OF cIFM_AL1342_Acyclic_Request;
END_VAR

IF Response.Port>0 THEN
	Port_Response[Response.Port]:=Response;
	Port_Response[Response.Port].Port:=0;
	
END_IF;

IF Port_Request[i+1].Port =16#FF THEN
	msgCounter:=msgCounter+1;
	Port_Request[i+1].Port:=TO_WORD(i+1);
	Port_Request[i+1].User_ID:=msgCounter;
	Request:=Port_Request[i+1];
	Acyclic_Request:=TRUE;
	
ELSE
	i:=(i+1) MOD 8;	
	Acyclic_Request:=FALSE;
END_IF;

END_FUNCTION_BLOCK

// Level_1_Devices/Analog_Control_UDFB
FUNCTION_BLOCK Analog_Control_UDFB
VAR_INPUT
	//Raw:	REAL;

	Alarm_Enable:BOOL:=TRUE;
	Latching:BOOL:=FALSE;
	Fault:BOOL:=FALSE;
	Online:BOOL:=TRUE;
END_VAR

VAR_OUTPUT
	//Status	:BYTE;
END_VAR

VAR_IN_OUT
	Device	:	Analog_Control_DUT;
END_VAR

VAR
	hihi: BOOL;
	hi: BOOL;
	lolo: BOOL;
	LO: BOOL;
	Alarm_Debounce: TON;
	deboune_Time: TIME;
	Alarm_Active: BOOL;
	Alarm_Debounce_ET: TIME;
	Alarm: BOOL;
	ALARM_2_0: BURKERT_OSCAT_BASIC.ALARM_2;
	F_TRIG_0: F_Trig;
	TON_0: TON;
END_VAR

VAR_TEMP
	EU_Range: REAL;
	Raw_Range: REAL;
	Corrected_Raw: REAL;
	Raw_Pct: REAL;
	EU_Scaled: REAL;
END_VAR
VAR // added by the converter: edge detectors and wires of the graphical bodies
    _w1 : BOOL;
END_VAR

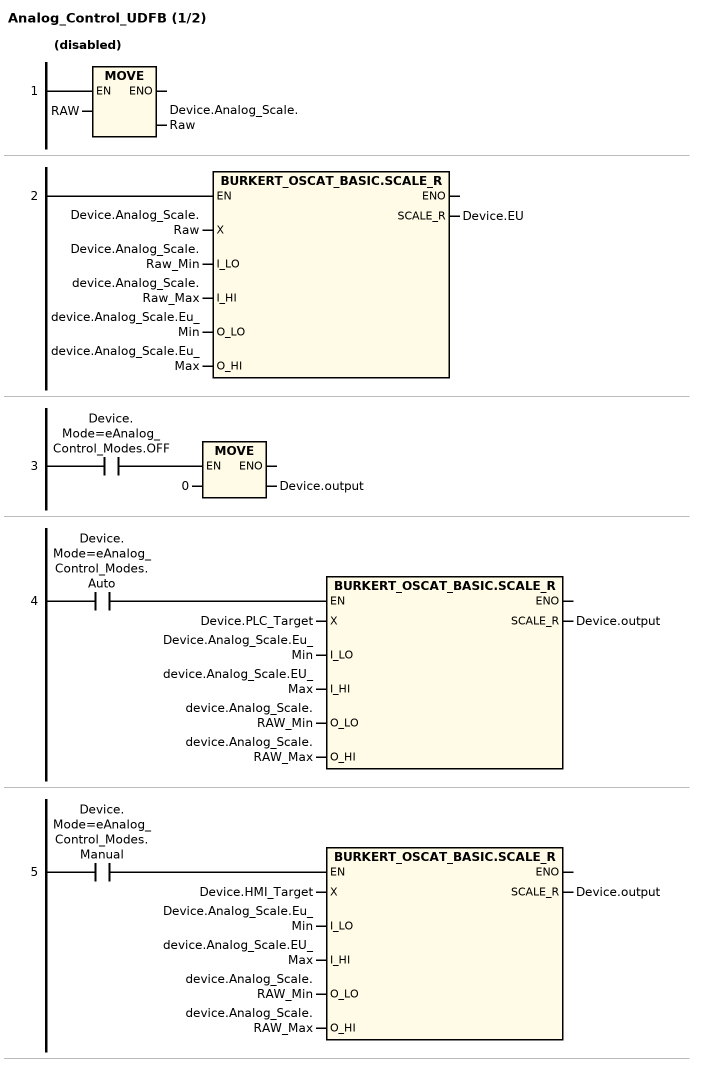
// NETWORK 1 (disabled)
// Device.Analog_Scale.Raw := RAW;

// NETWORK 2
Device.EU := BURKERT_OSCAT_BASIC.SCALE_R(X := Device.Analog_Scale.Raw, I_LO := Device.Analog_Scale.Raw_Min, I_HI := device.Analog_Scale.Raw_Max, O_LO := device.Analog_Scale.Eu_Min, O_HI := device.Analog_Scale.Eu_Max);

// NETWORK 3
IF Device.Mode=eAnalog_Control_Modes.OFF THEN Device.output := 0; END_IF

// NETWORK 4
IF Device.Mode=eAnalog_Control_Modes.Auto THEN
    Device.output := BURKERT_OSCAT_BASIC.SCALE_R(X := Device.PLC_Target, I_LO := Device.Analog_Scale.Eu_Min, I_HI := device.Analog_Scale.EU_Max, O_LO := device.Analog_Scale.RAW_Min, O_HI := device.Analog_Scale.RAW_Max);
END_IF

// NETWORK 5
IF Device.Mode=eAnalog_Control_Modes.Manual THEN
    Device.output := BURKERT_OSCAT_BASIC.SCALE_R(X := Device.HMI_Target, I_LO := Device.Analog_Scale.Eu_Min, I_HI := device.Analog_Scale.EU_Max, O_LO := device.Analog_Scale.RAW_Min, O_HI := device.Analog_Scale.RAW_Max);
END_IF

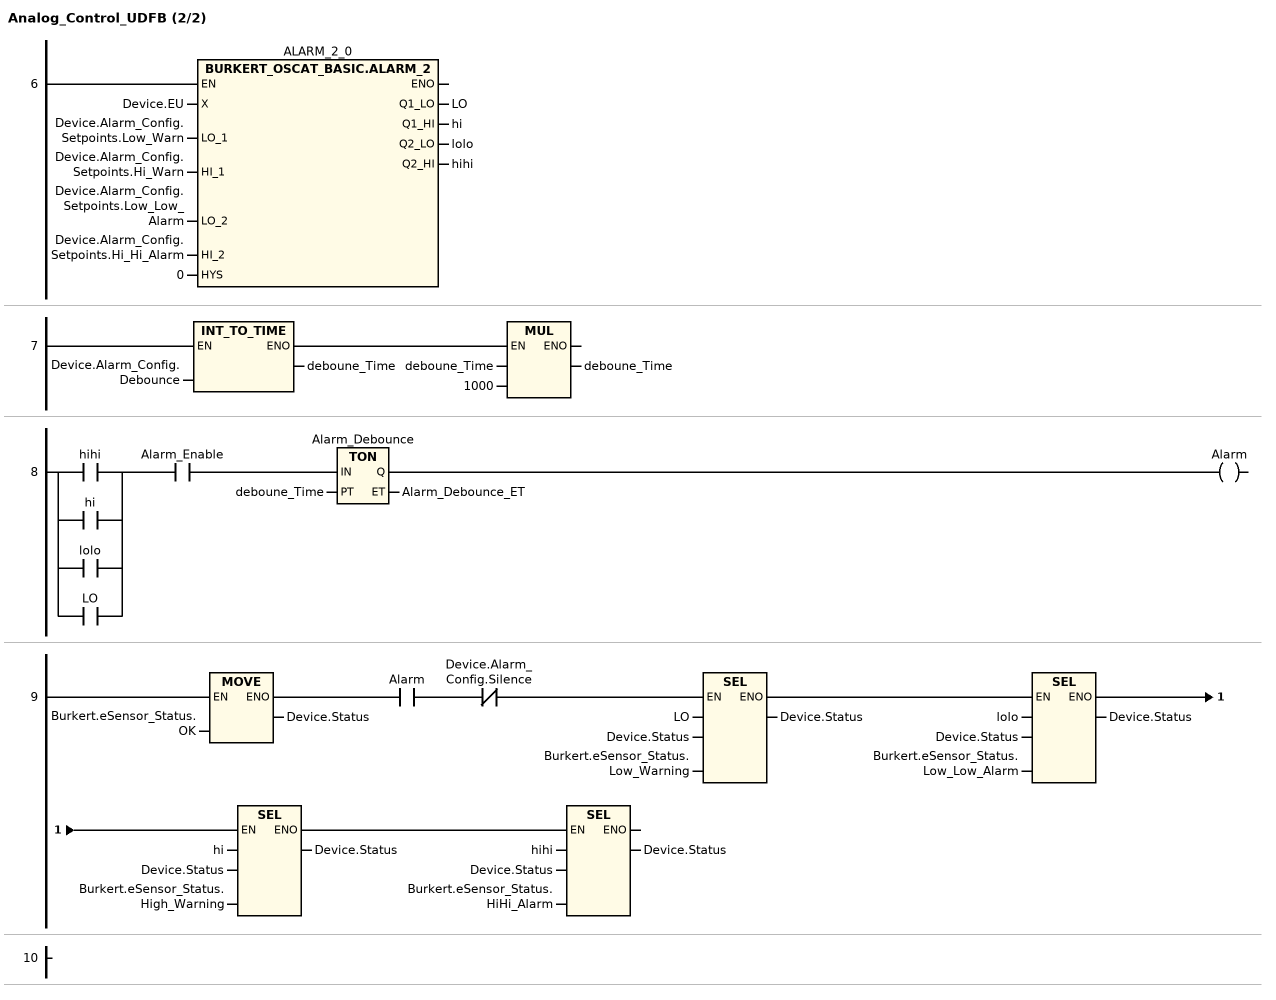
// NETWORK 6
ALARM_2_0(
    X := Device.EU,
    LO_1 := Device.Alarm_Config.Setpoints.Low_Warn,
    HI_1 := Device.Alarm_Config.Setpoints.Hi_Warn,
    LO_2 := Device.Alarm_Config.Setpoints.Low_Low_Alarm,
    HI_2 := Device.Alarm_Config.Setpoints.Hi_Hi_Alarm,
    HYS := 0,
    Q1_LO => LO,
    Q1_HI => hi,
    Q2_LO => lolo,
    Q2_HI => hihi); // BURKERT_OSCAT_BASIC.ALARM_2

// NETWORK 7
deboune_Time := INT_TO_TIME(Device.Alarm_Config.Debounce);
deboune_Time := deboune_Time * 1000;

// NETWORK 8
Alarm_Debounce(
    IN := (hihi OR hi OR lolo OR LO) AND Alarm_Enable,
    PT := deboune_Time,
    ET => Alarm_Debounce_ET); // TON
Alarm := Alarm_Debounce.Q;

// NETWORK 9
Device.Status := Burkert.eSensor_Status.OK;
_w1 := Alarm AND NOT Device.Alarm_Config.Silence;
IF _w1 THEN Device.Status := SEL(LO, Device.Status, Burkert.eSensor_Status.Low_Warning); END_IF
IF _w1 THEN Device.Status := SEL(lolo, Device.Status, Burkert.eSensor_Status.Low_Low_Alarm); END_IF
IF _w1 THEN Device.Status := SEL(hi, Device.Status, Burkert.eSensor_Status.High_Warning); END_IF
IF _w1 THEN Device.Status := SEL(hihi, Device.Status, Burkert.eSensor_Status.HiHi_Alarm); END_IF

// NETWORK 10

END_FUNCTION_BLOCK

// Level_1_Devices/Stack_Lights_4Way
FUNCTION_BLOCK Stack_Lights_4Way
VAR_INPUT
END_VAR
VAR_OUTPUT
	Red:BOOL;
	Yellow:BOOL;
	Green:BOOL;
	Horn:BOOL;
	
END_VAR
VAR
	
	GEN_PULSE_RED: Burkert_OSCAT_BASIC.GEN_PULSE;
	GEN_PULSE_Yellow: Burkert_OSCAT_BASIC.GEN_PULSE;
	GEN_PULSE_Green: Burkert_OSCAT_BASIC.GEN_PULSE;
	GEN_PULSE_Horn: Burkert_OSCAT_BASIC.GEN_PULSE;
END_VAR

VAR_IN_out
	Device:c4Way_Stack_Light;
END_VAR
VAR // added by the converter: edge detectors and wires of the graphical bodies
    _w1, _w2, _w3, _w4 : ANY;
END_VAR

GEN_PULSE_Yellow(
    ENQ := Device.Yellow.Flash_Rate_ms>500 AND Device.Yellow.ON,
    PTH := To_Time(Device.Yellow.Flash_Rate_ms),
    PTL := To_Time(Device.Yellow.Flash_Rate_ms)); // Burkert_OSCAT_BASIC.GEN_PULSE
GEN_PULSE_Green(
    ENQ := Device.Green.Flash_Rate_ms>500 AND Device.Green.ON,
    PTH := To_Time(Device.Green .Flash_Rate_ms),
    PTL := To_Time(Device.Green .Flash_Rate_ms)); // Burkert_OSCAT_BASIC.GEN_PULSE
GEN_PULSE_Horn(
    ENQ := Device.Horn.Flash_Rate_ms>500 AND Device.Horn.ON,
    PTH := To_Time(Device.Horn .Flash_Rate_ms),
    PTL := To_Time(Device.Horn .Flash_Rate_ms)); // Burkert_OSCAT_BASIC.GEN_PULSE
_w1 := Device.Horn.ON AND NOT GEN_PULSE_Horn.Q;
Horn := _w1;
_w2 := Device.Yellow.ON AND NOT GEN_PULSE_Yellow.Q;
Device.Yellow.Q := _w2;
Yellow := _w2;
_w3 := Device.Green.ON AND NOT GEN_PULSE_Green.Q;
Device.Green.Q := _w3;
Green := _w3;
GEN_PULSE_RED(
    ENQ := Device.RED.Flash_Rate_ms>500 AND Device.RED.ON,
    PTH := To_Time(Device.RED.Flash_Rate_ms),
    PTL := To_Time(Device.RED.Flash_Rate_ms)); // Burkert_OSCAT_BASIC.GEN_PULSE
_w4 := Device.RED.ON AND NOT GEN_PULSE_RED.Q;
Device.RED.Q := _w4;
Red := _w4;
Device.Horn.Q := _w1;

END_FUNCTION_BLOCK

// Level_2_Controls/Analog_Batch_Pump
FUNCTION_BLOCK Analog_Batch_Pump
VAR_INPUT
END_VAR
VAR_OUTPUT
	RUN:BOOL;
	Rev:BOOL;
	Speed:REAL;
END_VAR
VAR_IN_OUT
	Pump:cAnalog_Batch_Pump;
END_VAR
VAR
	Max_Volume:REAL;
	Min_Volume:REAL;
	TON_0: TON;
	TP_0: TP;
	TON_1: TON;
	F_TRIG_0: F_trig;
	Min_time:REAL;
	Max_Time:Real;
	New_Pump_Time: INT;
	lcl_Target:REAL;
	lcl_Seconds:REAL;
	Base_PCT: REAL;
	TON_2: TON;
	R_TRIG_0: R_trig;
	TP_1: TP;
	F_TRIG_1: F_trig;
	Cal_Value: REAL;
	RUN_REQ: BOOL;
	F_TRIG_2: F_Trig;
	TP_2: TP;
	CLK_PRG_0: BURKERT_OSCAT_BASIC.CLK_PRG;
	R_TRIG_1: R_trig;
END_VAR
VAR // added by the converter: edge detectors and wires of the graphical bodies
    _w1, _w6, _w9, _w10, _w11, _w12, _w13, _w14 : ANY;
    _w2, _w3, _w4, _w15 : REAL;
    _w5 : INT;
    _w7, _w8 : TIME;
END_VAR

